// TIA Portal V19 export
DATA_BLOCK "PID P-502 DB"   // DB173
{ S7_Optimized_Access := 'FALSE' }
   VAR
      PID_GAIN : Real;
      PID_I : Real;
      PID_D : Real;
      "P-502" : Struct
         "PV INPUT" : Real;
         "IN SETPOINT" : Real;
         "P-502 MAIN NEWOUT" : Real;
      END_STRUCT;
      SETPOINT : Real;
   END_VAR
BEGIN
END_DATA_BLOCK
